TYPE (* Complete ISOBUS UT scroll list configuration: geometry + operator controls, bundled for a single-struct FB interface *)
  (* Standard: 61499-2; Description: Copyright (c) 2026 Meisterschulen am Ostbahnhof This program and the accompanying materials are made available under the terms of the Eclipse Public License 2.0 which is available at https://www.eclipse.org/legal/epl-2.0/ SPDX-License-Identifier: EPL-2.0 *)
  (* Version 1.0, 2026-08-09, Franz Höpfinger, Meisterschulen am Ostbahnhof, initial API and implementation and/or initial documentation *)
  PACKAGE isobus::utils::scroll;
  IMPORT isobus::utils::scroll::ScrollObjectPool_S;
  IMPORT isobus::utils::scroll::ScrollControls_S;
  ScrollFull_S : STRUCT
    stGeometry : isobus::utils::scroll::ScrollObjectPool_S; (* List + scrollbar geometry and Change Child Position targets *)
    stControls : isobus::utils::scroll::ScrollControls_S; (* Operator control objects (6 buttons + direct-position input field) *)
  END_STRUCT;
END_TYPE
